// TwinCAT 3 PLC project Sample03
// ProgramVersion: 3.1.4022.4
// libraries:
//   Tc2_Standard, * (Beckhoff Automation GmbH)
//   Tc2_System, * (Beckhoff Automation GmbH)
//   Tc3_Module, * (Beckhoff Automation GmbH)
// project tree:
//   / ClassDiagram.TcCD (not stored), PlcTask.TcTTO
//   POUs/ FB_Decorator.TcPOU, FB_DecoratorCheese.TcPOU, FB_DecoratorSalami.TcPOU, FB_DecoratorTomato.TcPOU, FB_PizzaAmericanStyle.TcPOU, FB_PizzaItalianStyle.TcPOU, I_Pizza.TcIO, MAIN.TcPOU
// real-time tasks:
//   TASK PlcTask: cycle T#10ms, priority 20, ADS port 350

CONFIGURATION Sample03
    RESOURCE PLC ON TwinCAT3
        TASK PlcTask(INTERVAL := T#10ms, PRIORITY := 20);
        PROGRAM MAIN WITH PlcTask : MAIN;
    END_RESOURCE
END_CONFIGURATION

// ---- POUs/I_Pizza.TcIO
INTERFACE I_Pizza

METHOD GetDescription : STRING
VAR_INPUT
END_VAR
END_METHOD

METHOD GetPrice : LREAL
VAR_INPUT
END_VAR
END_METHOD

END_INTERFACE

// ---- POUs/MAIN.TcPOU
PROGRAM MAIN
VAR
	// Italian Pizza Margherita (via declaration)
	fbItalianStyle				: FB_PizzaItalianStyle;
	fbTomato					: FB_DecoratorTomato(fbItalianStyle, TRUE);
	fbCheese					: FB_DecoratorCheese(fbTomato);
	ipPizza						: I_Pizza := fbCheese;
	
	// Italian Pizza Margherita (via runtime)
	(* fbItalianStyle			: FB_PizzaItalianStyle;
	fbTomato					: FB_DecoratorTomato(0, FALSE);
	fbCheese					: FB_DecoratorCheese(0);
	ipPizza						: I_Pizza; *)
	
	bCreate						: BOOL;
	fPrice						: LREAL;
	sDescription				: STRING;
END_VAR

(* IF (bCreate) THEN
	bCreate := FALSE;
	fbTomato.ipDecorator := fbItalianStyle;
	fbCheese.ipDecorator := fbTomato;
	ipPizza := fbCheese;
END_IF *)

IF (ipPizza <> 0) THEN
	fPrice := ipPizza.GetPrice();
	sDescription := ipPizza.GetDescription();
END_IF

END_PROGRAM

// ---- POUs/FB_PizzaItalianStyle.TcPOU
FUNCTION_BLOCK PUBLIC FB_PizzaItalianStyle IMPLEMENTS I_Pizza
VAR_INPUT
END_VAR
VAR_OUTPUT
END_VAR
VAR
END_VAR

METHOD GetDescription : STRING
GetDescription := 'Pizza Italian Style:';
END_METHOD

METHOD GetPrice : LREAL
GetPrice := 4.5;
END_METHOD

END_FUNCTION_BLOCK

// ---- POUs/FB_DecoratorTomato.TcPOU
FUNCTION_BLOCK PUBLIC FB_DecoratorTomato EXTENDS FB_Decorator
VAR_INPUT
END_VAR
VAR_OUTPUT
END_VAR
VAR
	bWholefood		: BOOL;
END_VAR

PROPERTY PUBLIC bWholefoodProduct : BOOL
GET
bWholefoodProduct := THIS^.bWholefood;
END_GET
SET
THIS^.bWholefood := bWholefoodProduct;
END_SET
END_PROPERTY

METHOD FB_init : BOOL
VAR_INPUT
	bInitRetains		: BOOL; // if TRUE, the retain variables are initialized (warm start / cold start)
	bInCopyCode			: BOOL;  // if TRUE, the instance afterwards gets moved into the copy code (online change)
	ipSideOrder			: I_Pizza;
	bWholefoodProduct	: BOOL;
END_VAR
THIS^.bWholefood := bWholefoodProduct;
END_METHOD

METHOD GetDescription : STRING
IF (SUPER^.ipSideOrder <> 0) THEN
	GetDescription := CONCAT (SUPER^.ipSideOrder.GetDescription(), ' - Tomato');
	IF (THIS^.bWholefoodProduct) THEN
	GetDescription := CONCAT (GetDescription, ' (WholefoodProduct) ');
	END_IF
END_IF
END_METHOD

METHOD GetPrice : LREAL
IF (SUPER^.ipSideOrder <> 0) THEN
	GetPrice := SUPER^.ipSideOrder.GetPrice() + 0.9;
	IF (THIS^.bWholefood) THEN
		GetPrice := GetPrice + 0.3;
	END_IF
END_IF
END_METHOD

END_FUNCTION_BLOCK

// ---- POUs/FB_Decorator.TcPOU
FUNCTION_BLOCK PUBLIC FB_Decorator IMPLEMENTS I_Pizza
VAR_INPUT
END_VAR
VAR_OUTPUT
END_VAR
VAR
	ipSideOrder	: I_Pizza;
END_VAR

METHOD FB_init : BOOL
VAR_INPUT
	bInitRetains	: BOOL; // if TRUE, the retain variables are initialized (warm start / cold start)
	bInCopyCode		: BOOL;  // if TRUE, the instance afterwards gets moved into the copy code (online change)
	ipSideOrder		: I_Pizza;
END_VAR
THIS^.ipSideOrder := ipSideOrder;
END_METHOD

{warning 'add method implementation'}
METHOD GetDescription : STRING
END_METHOD

{warning 'add method implementation'}
METHOD GetPrice : LREAL
END_METHOD

PROPERTY PUBLIC ipDecorator : I_Pizza
GET
ipDecorator := THIS^.ipSideOrder;
END_GET
SET
THIS^.ipSideOrder := ipDecorator;
END_SET
END_PROPERTY

END_FUNCTION_BLOCK

// ---- POUs/FB_DecoratorCheese.TcPOU
FUNCTION_BLOCK PUBLIC FB_DecoratorCheese EXTENDS FB_Decorator
VAR_INPUT
END_VAR
VAR_OUTPUT
END_VAR
VAR
END_VAR

METHOD GetDescription : STRING
IF (SUPER^.ipSideOrder <> 0) THEN
	GetDescription := CONCAT (SUPER^.ipSideOrder.GetDescription(), ' - Cheese');
END_IF
END_METHOD

METHOD GetPrice : LREAL
IF (SUPER^.ipSideOrder <> 0) THEN
	GetPrice := SUPER^.ipSideOrder.GetPrice() + 1.1;
END_IF
END_METHOD

END_FUNCTION_BLOCK

// ---- POUs/FB_DecoratorSalami.TcPOU
FUNCTION_BLOCK PUBLIC FB_DecoratorSalami EXTENDS FB_Decorator
VAR_INPUT
END_VAR
VAR_OUTPUT
END_VAR
VAR
END_VAR

METHOD GetDescription : STRING
IF (SUPER^.ipSideOrder <> 0) THEN
	GetDescription := CONCAT (SUPER^.ipSideOrder.GetDescription(), ' - Salami');
END_IF
END_METHOD

METHOD GetPrice : LREAL
IF (SUPER^.ipSideOrder <> 0) THEN
	GetPrice := SUPER^.ipSideOrder.GetPrice() + 1.4;
END_IF
END_METHOD

END_FUNCTION_BLOCK

// ---- POUs/FB_PizzaAmericanStyle.TcPOU
FUNCTION_BLOCK PUBLIC FB_PizzaAmericanStyle IMPLEMENTS I_Pizza
VAR_INPUT
END_VAR
VAR_OUTPUT
END_VAR
VAR
END_VAR

METHOD GetDescription : STRING
GetDescription := 'Pizza American Style:';
END_METHOD

METHOD GetPrice : LREAL
GetPrice := 4.2;
END_METHOD

END_FUNCTION_BLOCK
